FUNCTION_BLOCK L6_FMS205 // EXTENDS L1_ModuleBase;


VAR_INPUT
	//IC		: BOOL := FALSE; 	// todos los módulos están en condiciones iniciales
//    Execute	: BOOL;
	fbPanel					: L5_Panel := (dr := dr);	
END_VAR

VAR_OUTPUT
//	Ready	: BOOL;
	//Failure	: BOOL;
	//Done	: BOOL;	
END_VAR	
VAR
	// Director, panel y tapas
	dr						: L1_Director;
	tapas					: L6_Tapas;
	
	// módulos de la FMS205
	mdAlimentador			: L3_Alimentador			:= (dr:=dr, ID := 1, Name := 'Alimentador');
	mdPickAndPlaceCarga 	: L3_PickAndPlace			:= (dr:=dr, ID := 2, Name := 'Carga');
	mdMedidorTapa			: L3_MedidorTapa			:= (dr:=dr, ID := 3, Name := 'Medidor');
	mdCaptadorInductivo 	: L3_CaptadorInductivo		:= (dr:=dr, ID := 4, Name := 'Inductivo');
	mdDetectorFotoelectrico : L3_DetectorFotoelectrico	:= (dr:=dr, ID := 5, Name := 'Fotoeléctrico');
	mdEvacuador			 	: L3_Evacuador				:= (dr:=dr, ID := 6, Name := 'Evacuador');
	mdPickAndPlaceDescarga 	: L3_PickAndPlace			:= (dr:=dr, ID := 7, Name := 'Descarga');
	mdPlatoDivisor			: L3_PlatoDivisor			:= (dr:=dr, ID := 8, Name := 'Plato');
	mdCinta					: L3_Cinta					:= (dr:=dr, ID := 9, Name := 'Cinta');
	
	// controladores a nivel estación
	ctrlF1Producir			: L4_FMS205_F1Producir_SFC; 
	ctrlF2SeqPrep			: L4_FMS205_F2SeqPrep_SFC;		
	ctrlF3SeqFin			: L4_FMS205_F3SeqFin_SFC;		
	ctrlF6Prueba			: L4_FMS205_F6Prueba_SFC;
END_VAR

METHOD InitialConditions : BOOL
(* La estación está en condiciones iniciales si cada módulo lo está *)
InitialConditions := (
		mdAlimentador.IC AND
		mdPickAndPlaceCarga.IC AND
		mdMedidorTapa.IC AND 
		mdCaptadorInductivo.IC AND
		mdDetectorFotoelectrico.IC AND
		mdEvacuador.IC AND
		mdPickAndPlaceDescarga.IC AND
		mdPlatoDivisor.IC AND
		mdCinta.IC )  OR dr.gmLocalHost;
END_METHOD

METHOD IsFailied : BOOL
IsFailied:=
	mdAlimentador.fbController.NumError <> 0 OR
	mdPickAndPlaceCarga.fbController.NumError <> 0 OR
	mdMedidorTapa.fbController.NumError <> 0 OR 
	mdCaptadorInductivo.fbController.NumError <> 0 OR
	mdDetectorFotoelectrico.fbController.NumError <> 0 OR
	mdEvacuador.fbController.NumError <> 0 OR
	mdPickAndPlaceDescarga.fbController.NumError <> 0 OR
	mdPlatoDivisor.fbController.NumError <> 0 OR
	mdCinta.fbController.NumError <> 0 OR
	ctrlF1Producir.NumError <> 0 OR
	ctrlF2SeqPrep.NumError <> 0 OR
	ctrlF3SeqFin.NumError <> 0 OR
	ctrlF6Prueba.NumError <> 0;
END_METHOD

METHOD IsPaused : BOOL
VAR_INPUT
END_VAR
IsPaused := 
		mdAlimentador.fbController.IsPaused() AND
		mdPickAndPlaceCarga.fbController.IsPaused() AND
		mdMedidorTapa.fbController.IsPaused() AND 
		mdCaptadorInductivo.fbController.IsPaused() AND
		mdDetectorFotoelectrico.fbController.IsPaused() AND
		mdEvacuador.fbController.isPaused() AND
		mdPickAndPlaceDescarga.fbController.IsPaused() AND
		mdPlatoDivisor.fbController.IsPaused() AND
		mdCinta.fbController.IsPaused() AND
		ctrlF1Producir.IsPaused() AND
		ctrlF2SeqPrep.IsPaused() AND
		ctrlF3SeqFin.IsPaused() AND
		ctrlF6Prueba.IsPaused();
END_METHOD

METHOD IsReady : BOOL
VAR_INPUT
	gmMode	: L1_GEMMA;
END_VAR
CASE gmMode OF
	
	L1_GEMMA.F1ProduccionNormal,
	L1_GEMMA.F6Probando: 
		IsReady := (
			mdAlimentador.fbController.Ready AND
			mdPickAndPlaceCarga.fbController.Ready AND
			mdMedidorTapa.fbController.Ready AND 
			mdCaptadorInductivo.fbController.Ready AND
			mdDetectorFotoelectrico.fbController.Ready AND
			mdEvacuador.fbController.Ready AND
			mdPickAndPlaceDescarga.fbController.Ready AND
			mdPlatoDivisor.fbController.Ready AND
			mdCinta.fbController.Ready);
			
	 L1_GEMMA.F2SecuenciaPreparacion: 
		IsReady := (
			mdMedidorTapa.fbController.Ready AND 
			mdCaptadorInductivo.fbController.Ready AND
			mdDetectorFotoelectrico.fbController.Ready AND
			mdPlatoDivisor.fbController.Ready);
	
	L1_GEMMA.F3SecuenciaFinalizacion: 
		IsReady := (
			mdEvacuador.fbController.Ready AND
			mdPlatoDivisor.fbController.Ready);
END_CASE
END_METHOD

METHOD ManageErrors : BOOL
mdAlimentador.fbController.ResetError();
mdAlimentador.fbController.ResetError();
mdPickAndPlaceCarga.fbController.ResetError();
mdMedidorTapa.fbController.ResetError();
mdCaptadorInductivo.fbController.ResetError();
mdDetectorFotoelectrico.fbController.ResetError();
mdEvacuador.fbController.ResetError();
mdPickAndPlaceDescarga.fbController.ResetError();
mdPlatoDivisor.fbController.ResetError();
mdCinta.fbController.ResetError();
ctrlF1Producir.ResetError();
ctrlF2SeqPrep.ResetError();
ctrlF3SeqFin.ResetError();
ctrlF6Prueba.ResetError();
END_METHOD

METHOD ProcessCycle : BOOL
// calcular consignas en función del panel y del modo Gemma

fbPanel.ProcessCycle(dr:=dr, gmModeActual := dr.gmModeActual, tmReinicio := dr.tmTiempoReinicio); 

// controlar el flujo a nivel de la estación
CASE dr.gmModeActual OF
	L1_GEMMA.A6Inicializando:
		tapas.A1Inicializar(DebePreparar:=dr.cnF2_Preparar);		
		
	L1_GEMMA.A1ParadaInicial:
		; // esperar a que se pida hacer altgo
		
	L1_GEMMA.F4VerificacionSinOrden: 
		IF fbPanel.swF4_Avanza THEN		
			mdCinta.Avanza();				// si se pulsa avanzar activar RUN y desactivar REV
		ELSIF fbPanel.swF4_Retroc THEN
			mdCinta.Retrocede();			// si se pulsa retrocede activar RUN y REV
		END_IF

	L1_GEMMA.A2ParaFinCiclo,
	L1_GEMMA.F1ProduccionNormal:
		ctrlF1Producir.IC 				:= InitialConditions();
		IF ctrlF1Producir.Ready AND NOT dr.EndBatch THEN
			ctrlF1Producir.Execute		:= TRUE;
			ctrlF1Producir.Ack			:= FALSE;
			tapas.A2InicioCiclo();
			mdPickAndPlaceCarga.Mover 	:= tapas.ExeCarga;
			mdEvacuador.Evacuar 		:= tapas.ExeEvacu;
			mdPickAndPlaceDescarga.Mover:= tapas.ExeDesca;
		ELSIF ctrlF1Producir.Done THEN
			ctrlF1Producir.Execute		:= FALSE;
			ctrlF1Producir.Ack			:= TRUE;			
		END_IF
		ctrlF1Producir(Alime:=mdAlimentador, Carga:=mdPickAndPlaceCarga, Medid:=mdMedidorTapa, Fotoe:=mdDetectorFotoelectrico, 
			Induc:=mdCaptadorInductivo, Evacu:=mdEvacuador,	Desca:=mdPickAndPlaceDescarga, Plato:=mdPlatoDivisor, Cinta:=mdCinta);

	L1_GEMMA.F2SecuenciaPreparacion:		
		IF ctrlF2SeqPrep.Ready THEN
			ctrlF2SeqPrep.Execute 			:= TRUE; // ctrlF2SeqPrep.Ready;
			ctrlF2SeqPrep.Ack				:= FALSE;
			ctrlF2SeqPrep.cnF2_Preparar		:= dr.cnF2_Preparar;
			ctrlF2SeqPrep.TapasOk 			:= FALSE;
		ELSIF ctrlF2SeqPrep.InitTapas THEN
			tapas.A2InicioCiclo();		
			ctrlF2SeqPrep.TapasOk 			:= TRUE;	
		ELSIF ctrlF2SeqPrep.Done THEN
			dr.cnF2_Preparar 				:= FALSE;
			ctrlF2SeqPrep.Execute 			:= FALSE;
			ctrlF2SeqPrep.Ack				:= TRUE;
		ELSE
			ctrlF2SeqPrep.IC				:= InitialConditions();
		END_IF
		ctrlF2SeqPrep(Medid:=mdMedidorTapa, Fotoe:=mdDetectorFotoelectrico,	Induc:=mdCaptadorInductivo, Plato:=mdPlatoDivisor);		

	L1_GEMMA.F3SecuenciaFinalizacion:
		IF ctrlF3SeqFin.Ready THEN
			ctrlF3SeqFin.Execute 			:= TRUE; // ctrlF3SeqFin.Ready;
			ctrlF3SeqFin.Ack				:= FALSE;
			ctrlF3SeqFin.cnF3_Finalizar		:= dr.cnF3_Finalizar;
			ctrlF3SeqFin.TapasOk			:= FALSE;
		ELSIF ctrlF3SeqFin.InitTapas THEN
			tapas.A2InicioCiclo();		
			mdEvacuador.Evacuar				:= tapas.ExeEvacu;
			ctrlF3SeqFin.TapasOk 			:= TRUE;
		ELSIF ctrlF3SeqFin.Done THEN
			dr.cnF3_Finalizar 				:= FALSE;
			ctrlF3SeqFin.Execute 			:= FALSE;
			ctrlF3SeqFin.Ack				:= TRUE;
		ELSE
			ctrlF3SeqFin.IC					:= InitialConditions();
		END_IF
		ctrlF3SeqFin(Evacu:=mdEvacuador, Plato:=mdPlatoDivisor);

	L1_GEMMA.F6Probando:
		IF ctrlF6Prueba.Ready THEN
			ctrlF6Prueba.Execute 			:= TRUE;
			ctrlF6Prueba.Ack				:= FALSE; // ctrlF6Prueba.Done;  //IsReady(gmMode:=L1_GEMMA.F6Probando);
			tapas.A2InicioCiclo();		
			mdPickAndPlaceCarga.Mover 		:= tapas.ExeCarga;
			mdEvacuador.Evacuar 			:= tapas.ExeEvacu;
			mdPickAndPlaceDescarga.Mover	:= tapas.ExeDesca;
		ELSIF ctrlF6Prueba.Done THEN
			ctrlF6Prueba.Ack				:= TRUE; // ctrlF6Prueba.Done;  //IsReady(gmMode:=L1_GEMMA.F6Probando);
			ctrlF6Prueba.Execute 			:= FALSE;			
		ELSE
			ctrlF6Prueba.IC					:= InitialConditions();
		END_IF			
		ctrlF6Prueba(Alime:=mdAlimentador, Carga:=mdPickAndPlaceCarga, Medid:=mdMedidorTapa, Fotoe:=mdDetectorFotoelectrico, 
			Induc:=mdCaptadorInductivo, Evacu:=mdEvacuador,	Desca:=mdPickAndPlaceDescarga, Plato:=mdPlatoDivisor, Cinta:=mdCinta);

	L1_GEMMA.F5VerificacionOrdenada: 		// tener en cuenta las consignas relacionadas con F5 		
		mdAlimentador.Execute          		:= fbPanel.swF5_Ejecutar AND fbPanel.swF5_Alimentar;
		mdPickAndPlaceCarga.Execute    		:= fbPanel.swF5_Ejecutar AND fbPanel.swF5_Cargar;
		mdMedidorTapa.Execute          		:= fbPanel.swF5_Ejecutar AND fbPanel.swF5_Medir;
		mdDetectorFotoelectrico.Execute		:= fbPanel.swF5_Ejecutar AND fbPanel.swF5_Claridad;
		mdCaptadorInductivo.Execute    		:= fbPanel.swF5_Ejecutar AND fbPanel.swF5_Material;
		mdEvacuador.Execute            		:= fbPanel.swF5_Ejecutar AND fbPanel.swF5_Evacuar;
		mdPickAndPlaceDescarga.Execute		:= fbPanel.swF5_Ejecutar AND fbPanel.swF5_Descargar;
		mdPlatoDivisor.Execute       		:= fbPanel.swF5_Ejecutar AND fbPanel.swF5_Girar;
		mdCinta.Situar						:= fbPanel.swF5_Situar;
		mdCinta.Transferir					:= fbPanel.swF5_Transferir;
		mdCinta.Execute						:= fbPanel.swF5_Ejecutar AND (fbPanel.swF5_Situar OR fbPanel.swF5_Transferir);		
		mdPickAndPlaceCarga.Mover	    	:= TRUE; 
		mdEvacuador.Evacuar 				:= TRUE; 
		mdPickAndPlaceDescarga.Mover		:= TRUE; 
		mdAlimentador.Ack               	:= fbPanel.swF5_Ack AND fbPanel.swF5_Alimentar;
		mdPickAndPlaceCarga.Ack         	:= fbPanel.swF5_Ack AND fbPanel.swF5_Cargar;
		mdMedidorTapa.Ack               	:= fbPanel.swF5_Ack AND fbPanel.swF5_Medir;
		mdDetectorFotoelectrico.Ack			:= fbPanel.swF5_Ack AND fbPanel.swF5_Claridad;
		mdCaptadorInductivo.Ack         	:= fbPanel.swF5_Ack AND fbPanel.swF5_Material;
		mdEvacuador.Ack                 	:= fbPanel.swF5_Ack AND fbPanel.swF5_Evacuar;
		mdPickAndPlaceDescarga.Ack      	:= fbPanel.swF5_Ack AND fbPanel.swF5_Descargar;
		mdPlatoDivisor.Ack              	:= fbPanel.swF5_Ack AND fbPanel.swF5_Girar;
		mdCinta.Ack							:= fbPanel.swF5_Ack AND (fbPanel.swF5_Situar OR fbPanel.swF5_Transferir);
		
						
	L1_GEMMA.A3ParadaEstado, 
	L1_GEMMA.A4ParadaObtenida:
		dr.IsPaused := IsPaused(); // esperar la puesta en marcha o reanudar tras parada

	L1_GEMMA.D2TratamientoFallos:
		dr.Failure 		:= IsFailied(); // redundante. ManageErrors(); // esperar a que el usuario arregle el error
		
	L1_GEMMA.A5PreparandoTrasFallo:
		ManageErrors();;
		
 
END_CASE




ctrlF1Producir.ProcessCycle(dr.gmModeActual);
ctrlF2SeqPrep.ProcessCycle(dr.gmModeActual);
ctrlF3SeqFin.ProcessCycle(dr.gmModeActual);
ctrlF6Prueba.ProcessCycle(dr.gmModeActual);

// ejecutar el ciclo de cada uno de los módulos
mdAlimentador.ProcessCycle				(dr:=dr, tapas:=tapas);
mdPickAndPlaceCarga.ProcessCycle		(dr:=dr, tapas:=tapas);
mdMedidorTapa.ProcessCycle				(dr:=dr, tapas:=tapas);	
mdDetectorFotoelectrico.ProcessCycle	(dr:=dr, tapas:=tapas);
mdCaptadorInductivo.ProcessCycle		(dr:=dr, tapas:=tapas);
mdEvacuador.ProcessCycle				(dr:=dr, tapas:=tapas);
mdPickAndPlaceDescarga.ProcessCycle		(dr:=dr, tapas:=tapas);
mdPlatoDivisor.ProcessCycle				(dr:=dr, tapas:=tapas);
mdCinta.ProcessCycle					(dr:=dr, tapas:=tapas);

// actualizar la interfaz de usuario
tapas.Actualizar();
tapas.Animar(PlatoActivo := NOT mdPlatoDivisor.fbController.Ready);


dr.IC			:= InitialConditions();
dr.Failure 		:= IsFailied();
dr.EndCycle 	:= ctrlF1Producir.Done;
dr.EndBatch 	:= tapas.ResReal >= tapas.ReqNumero;
dr.ProcessCycle();
END_METHOD

END_FUNCTION_BLOCK

(* stored: Version 1.1.0.1, ProductVersion 3.1.4024.11
   POU L6_FMS205: Id {a261f573-1402-443e-9bab-e88e0bf02070}, SpecialFunc None
   Method InitialConditions: Id {6c17034c-aab7-41fb-b0b6-e85a6db67498}
   Method IsFailied: Id {c00d0657-d8cd-4b4b-a9ee-6be440092cb6}
   Method IsPaused: Id {63c7f49b-23e4-43c3-ac69-584bc16d9aec}
   Method IsReady: Id {22492767-8d7d-4c2f-892d-876b7dde965e}
   Method ManageErrors: Id {fa49f856-5c55-4bc1-adc6-7253af1cd7df}
   Method ProcessCycle: Id {02e4c75f-69e3-444f-8a2e-ecad65532e26} *)
